Staubli VAL3: GenericApp.pjx

Parameters version=s7.0 stackSize=5000 millimeterUnit=true
Program file=init.pgx
Program file=start.pgx
Program file=stop.pgx
Data file=GenericApp.dtx
Library alias=mot path=Disk://Tracking/Motion/Motion.pjx
